PROGRAM State_Machine
VAR
	//Data Send 2 FEC
		DataSend2FEC 		AT %Q*		: data_16real;
		
	//Data Received
		DataReceived AT %I*: data_16real;

	//Current state of FLC
		CurrentState : eCurrentState;

		// Current State of FEC
		FEC_CurrState : eFEC_CurrState;
		
		P_mod_ref : REAL;
		Q_mod_ref : REAL;
		
		RampDown : REAL := 1;
	wAutoManCtl: INT;
	
	Hugo :REAL;
	Hugo1 : INT;
	Hugo2 : INT;
	Hugo3: INT;
	Hugo4: INT;
	
			
	EtherCATHeartBeat : DINT;
	CounterCommFailure : INT;
	
	
	TIMER_TIMEOUT:TON;	// Timer for enabling TLC communication
	TS_TIMEOUT: TIME;
	Counter_TimeOUT : INT;
	TS_WARNING: TIME;
	EmergencyStop_TimeOut	:	BOOL;
	Counter_TimeOUT_2	:	INT;
END_VAR

// Protection for EtherCAT
	IF Communications.EtherCAT_Inputs_DINT.Heartbeat = EtherCATHeartBeat THEN
		CounterCommFailure := CounterCommFailure + 1;
			IF CounterCommFailure > 500 THEN
				Communications.EtherCAT_Inputs_DINT.Command := 0;
				GlobalVar.CommunicationFailureEtherCAT := TRUE;
				Communications.EtherCAT_Variables.WarningLog.Bits.EtherCAT_Failure := TRUE;
				CounterCommFailure := 0;
			END_IF
	ELSE
		GlobalVar.CommunicationFailureEtherCAT := FALSE;
		Communications.EtherCAT_Variables.WarningLog.Bits.EtherCAT_Failure := FALSE;
		CounterCommFailure := 0;
	END_IF
	EtherCATHeartBeat := Communications.EtherCAT_Inputs_DINT.Heartbeat;
// End of protection for EtherCAT


{IF defined (JEMA)}
	Hugo1 := 1;
	Mapping_ModbusReadRegisters(ADR(GlobalVar.ScaledModRead),ADR(Communications.EtherCAT_Monitor_Variables),ADR(Communications.EtherCAT_Variables));	
	Mapping_ModbusWriteRegisters(ADR(GlobalVar.ModWrite),ADR(Communications.EtherCAT_Inputs));
{ELSE}	
	Hugo1 := 2;
	GlobalVar.ModWrite.wAutoManCtl := REAL_TO_UINT(Communications.EtherCAT_Inputs.Command);
{END_IF}

//Rempaing from DINT To REAL and from REAL TO DINT.
Remap_EtherCAT_Variables(ADR(Communications.EhterCAT_Parameters_DINT),
						ADR(Communications.EtherCAT_EAP_Parameters_DINT),
						ADR(Communications.EtherCAT_Inputs_DINT),
						ADR(Communications.EtherCAT_Monitor_Variables_DINT),
						ADR(Communications.EhterCAT_Parameters),
						ADR(Communications.EtherCAT_EAP_Parameters),
						ADR(Communications.EtherCAT_Inputs),
						ADR(Communications.EtherCAT_Monitor_Variables));
			
//Read state machine of the Front End Controller.
		{IF defined (JEMA)}
			Hugo2 := 1;
			//Read state machine OF the Front End Controller.
			IF GlobalVar.ModRead.CtrlPriority = 1 THEN
				FEC_CurrState := UINT_TO_INT(GlobalVar.ModRead.fbOpMode);
			ELSE
				FEC_CurrState := 2;
			END_IF
		{ELSE}	
			Hugo2 := 2;
			FEC_CurrState := UINT_TO_INT(GlobalVar.ModRead.DerOpMode);
		{END_IF}
		
	IF GlobalVar.CommunicationFailureModbus = 1 THEN
		FEC_CurrState := 0;
	END_IF
					
//ALARMS FROM THE POWER CONVERTER.		

{IF defined (JEMA)}
	Hugo3 := 3;
	IF GlobalVar.ModRead.GrAlm0 > 0 THEN
		FEC_CurrState := 0;				
	END_IF
	IF GlobalVar.ModRead.GrAlm1 > 0 THEN
		FEC_CurrState := 0;				
	END_IF
	IF GlobalVar.ModRead.GrAlm2 > 0 THEN
		FEC_CurrState := 0;				
	END_IF
	IF GlobalVar.ModRead.GrAlm3 > 0 THEN
		FEC_CurrState := 0;				
	END_IF
	IF GlobalVar.ModRead.GrAlm4 > 0 THEN
		FEC_CurrState := 0;				
	END_IF
{ELSE}	
	Hugo3 := 2;
{END_IF}

//State Machine - First Level Controller
	CASE FEC_CurrState OF
		eFEC_CurrState.FEC_OFF:
			CurrentState := eCurrentState.OFF;
			GlobalVar.ModbusSPC_Enable := FALSE;
			GlobalVar.EAP_SPC_Enable := FALSE;
			
		eFEC_CurrState.FEC_STANDBY:
			CurrentState := eCurrentState.STANDBY;
			GlobalVar.ModbusSPC_Enable := FALSE;
			GlobalVar.EAP_SPC_Enable := FALSE;
			
		eFEC_CurrState.FEC_MANUAL:
			CurrentState := eCurrentState.STANDBY;
			GlobalVar.ModbusSPC_Enable := FALSE;
			GlobalVar.EAP_SPC_Enable := FALSE;
			
		eFEC_CurrState.FEC_AVG_PWR_CTR:
			CurrentState := eCurrentState.AVG_PWR_CTR;
			GlobalVar.ModbusSPC_Enable := TRUE;
			GlobalVar.EAP_SPC_Enable := FALSE;
			
		eFEC_CurrState.FEC_INST_PWR_CTR:
			CurrentState := eCurrentState.INST_PWR_CTR;
			GlobalVar.ModbusSPC_Enable := FALSE;
			
			IF GlobalVar.CommunicationFailureEtherCAT = FALSE THEN
				GlobalVar.EAP_SPC_Enable := TRUE;
			ELSE
				GlobalVar.EAP_SPC_Enable := FALSE;
			END_IF
	ELSE
		CurrentState := eCurrentState.STANDBY;	
	END_CASE
	
	{IF defined (JEMA)}
		Hugo := 1;
		Mapping_Monitoring_Variables(GlobalVar.ScaledModRead,ADR(Communications.EtherCAT_Monitor_Variables),ADR(Communications.EtherCAT_Variables));
	{ELSE}
		Hugo := 2;
		Mapping_Monitoring_Variables_ABG(GlobalVar.ModRead,ADR(Communications.EtherCAT_Monitor_Variables),ADR(Communications.EtherCAT_Variables));
	{END_IF}
	

//////////Alarms/Warnings of our system
	TS_TIMEOUT := STRING_TO_TIME(INSERT('T#ms','1000',2));
	TIMER_TIMEOUT(IN:= NOT TIMER_TIMEOUT.Q, PT:= TS_TIMEOUT);
	
	IF GlobalVar.CommunicationFailureModbus = TRUE THEN
		Communications.EtherCAT_Variables.WarningLog.Bits.ModbusComm_FLC_PCS := TRUE;	
	ELSE
		Communications.EtherCAT_Variables.WarningLog.Bits.ModbusComm_FLC_PCS := FALSE;	
	END_IF
	

	IF (Communications.EtherCAT_Inputs.Command <> Communications.EtherCAT_Variables.Status) AND  Communications.EtherCAT_Inputs.Command <> 100 THEN
		IF TIMER_TIMEOUT.Q THEN
			Counter_TimeOUT := Counter_TimeOUT + 1;
		END_IF
		IF Counter_TimeOUT = 120 THEN
			Communications.EtherCAT_Variables.WarningLog.Bits.CommandTimeout := TRUE; 
			Counter_TimeOUT := 0;
		END_IF
	ELSE 
		IF TIMER_TIMEOUT.Q THEN
			Counter_TimeOUT_2 := Counter_TimeOUT_2 + 1;
		END_IF
		
		IF Counter_TimeOUT_2 = 300 THEN
			Communications.EtherCAT_Variables.WarningLog.Bits.CommandTimeout := FALSE; 
			Counter_TimeOUT_2 := 0;
		END_IF	
		Counter_TimeOUT := 0;
	END_IF
	
	IF Communications.EtherCAT_Monitor_Variables.Vrmsa > Communications.EhterCAT_Parameters.CommonBlock_Params.NominalVoltage*1.4 THEN
		Communications.EtherCAT_Variables.WarningLog.Bits.OverVoltage := TRUE;
	ELSE
		Communications.EtherCAT_Variables.WarningLog.Bits.OverVoltage := FALSE;
	END_IF
	
	IF Communications.EtherCAT_Monitor_Variables.Vrmsa < Communications.EhterCAT_Parameters.CommonBlock_Params.NominalVoltage*0.5 THEN
		Communications.EtherCAT_Variables.WarningLog.Bits.UnderVoltage := TRUE;
	ELSE
		Communications.EtherCAT_Variables.WarningLog.Bits.UnderVoltage := FALSE;
	END_IF
	
	IF Communications.EtherCAT_Monitor_Variables.Irmsa > Communications.EhterCAT_Parameters.CommonBlock_Params.NominalPower/(3*(Communications.EhterCAT_Parameters.CommonBlock_Params.NominalVoltage+1)) THEN
		Communications.EtherCAT_Variables.WarningLog.Bits.OverCurrent := TRUE;
	ELSE
		Communications.EtherCAT_Variables.WarningLog.Bits.OverCurrent := FALSE;
	END_IF
	
	IF Communications.EtherCAT_Monitor_Variables.GridFre*0.1591549430918 > (Communications.EhterCAT_Parameters.CommonBlock_Params.NominalFreq +  Communications.EhterCAT_Parameters.CommonBlock_Params.NominalFreq*0.02) THEN
		Communications.EtherCAT_Variables.WarningLog.Bits.OverFrequency := TRUE;
	ELSE
		Communications.EtherCAT_Variables.WarningLog.Bits.OverFrequency := FALSE;
	END_IF
	
	IF Communications.EtherCAT_Monitor_Variables.GridFre*0.1591549430918 < (Communications.EhterCAT_Parameters.CommonBlock_Params.NominalFreq - Communications.EhterCAT_Parameters.CommonBlock_Params.NominalFreq*0.02) THEN
		Communications.EtherCAT_Variables.WarningLog.Bits.UnderFrequency := TRUE;
	ELSE
		Communications.EtherCAT_Variables.WarningLog.Bits.UnderFrequency := FALSE;
	END_IF
	
	IF Communications.PowerOfService.InertiaEmulationP_Service > Communications.EhterCAT_Parameters.InertiaEmulation_Params.PowerLimit_Inertia THEN
		Communications.EtherCAT_Variables.WarningLog.Bits.Inertia_Overrange := TRUE;
	ELSE
		Communications.EtherCAT_Variables.WarningLog.Bits.Inertia_Overrange := FALSE;
	END_IF 
	
	IF Communications.PowerOfService.FrequencyRegulationP_Service > Communications.EhterCAT_Parameters.FrequencyRegulation_Params.PowerLimit_Freq THEN
		Communications.EtherCAT_Variables.WarningLog.Bits.Frequency_Overrange := TRUE;
	ELSE
		Communications.EtherCAT_Variables.WarningLog.Bits.Frequency_Overrange := FALSE;
	END_IF
	
	IF Communications.PowerOfService.VoltageRegulationQ_Service > Communications.EhterCAT_Parameters.VoltageRegulation_Params.PowerLimit_Voltage THEN
		Communications.EtherCAT_Variables.WarningLog.Bits.VoltReg_Overrange := TRUE;
	ELSE
		Communications.EtherCAT_Variables.WarningLog.Bits.VoltReg_Overrange := FALSE;
	END_IF
	
	IF Communications.PowerOfService.ModalFreqAttP_Service > Communications.EhterCAT_Parameters.ModalFrequency_Params.PowerLimit_ModalFreq THEN
		Communications.EtherCAT_Variables.WarningLog.Bits.ModFreq_Overrange := TRUE;
	ELSE
		Communications.EtherCAT_Variables.WarningLog.Bits.ModFreq_Overrange := FALSE;
	END_IF
	
	IF Communications.EtherCAT_Monitor_Variables.BatSoc > 80 THEN
		Communications.EtherCAT_Variables.WarningLog.Bits.Battery_80Perc := TRUE;
	ELSE
		Communications.EtherCAT_Variables.WarningLog.Bits.Battery_80Perc := FALSE;
	END_IF
	
	IF Communications.EtherCAT_Monitor_Variables.BatSoc < 20 THEN
		Communications.EtherCAT_Variables.WarningLog.Bits.Battery_20Perc := TRUE;
	ELSE
		Communications.EtherCAT_Variables.WarningLog.Bits.Battery_20Perc := FALSE;
	END_IF
	
	
	/////////////////////Critical warnings
	IF Communications.EtherCAT_Variables.WarningLog.Bits.ModbusComm_FLC_PCS = TRUE THEN
		Communications.EtherCAT_Inputs.Command := 0;
		Communications.EtherCAT_Variables.Status := 0;
	END_IF
	
	IF Communications.EtherCAT_Variables.WarningLog.Bits.CommandTimeout = TRUE THEN
		Communications.EtherCAT_Inputs.Command := 0;
	END_IF
	
	IF Communications.EtherCAT_Variables.WarningLog.Bits.EtherCAT_Failure = TRUE THEN
		Communications.EtherCAT_Inputs.Command := 0;
		Communications.EtherCAT_Variables.Status := 0;
	END_IF

END_PROGRAM

(* stored: Version 1.1.0.1, ProductVersion 3.1.4024.11
   POU State_Machine: Id {f2669584-332a-4cf9-b7b0-658d596d50a2}, SpecialFunc None *)
